PROGRAM r_Gestion_Actionneurs_TOR
VAR
	XV_Alim_Douche: Registre_V1;
	XV_Alim_Douchette: Registre_V1;
	XV_Alim_Lavabo: Registre_V1;
	XV_Vid_Douche: Registre_V1;
	XV_Vid_Lavabo: Registre_V1;
	XV_Electrovanne_Douche: Registre_V1;
	XV_Electrovanne_Lavabo: Registre_V1;
	Prise_Cabine: Prise;
	XV_Vanne_Souf_Bas_Deb: Registre_V1;
	XV_Vanne_Ext_Bas_Deb: Registre_V1;
	Reg_Etanche_Souf: Registre_V1;
	XV_Alim_NEP: Registre_V1;
	Y_Verin_WC_GV: Registre_V1;
	Y_Verin_WC_PV: Registre_V1;
	Gestion_EA_WC: Sontay_4RM;
END_VAR

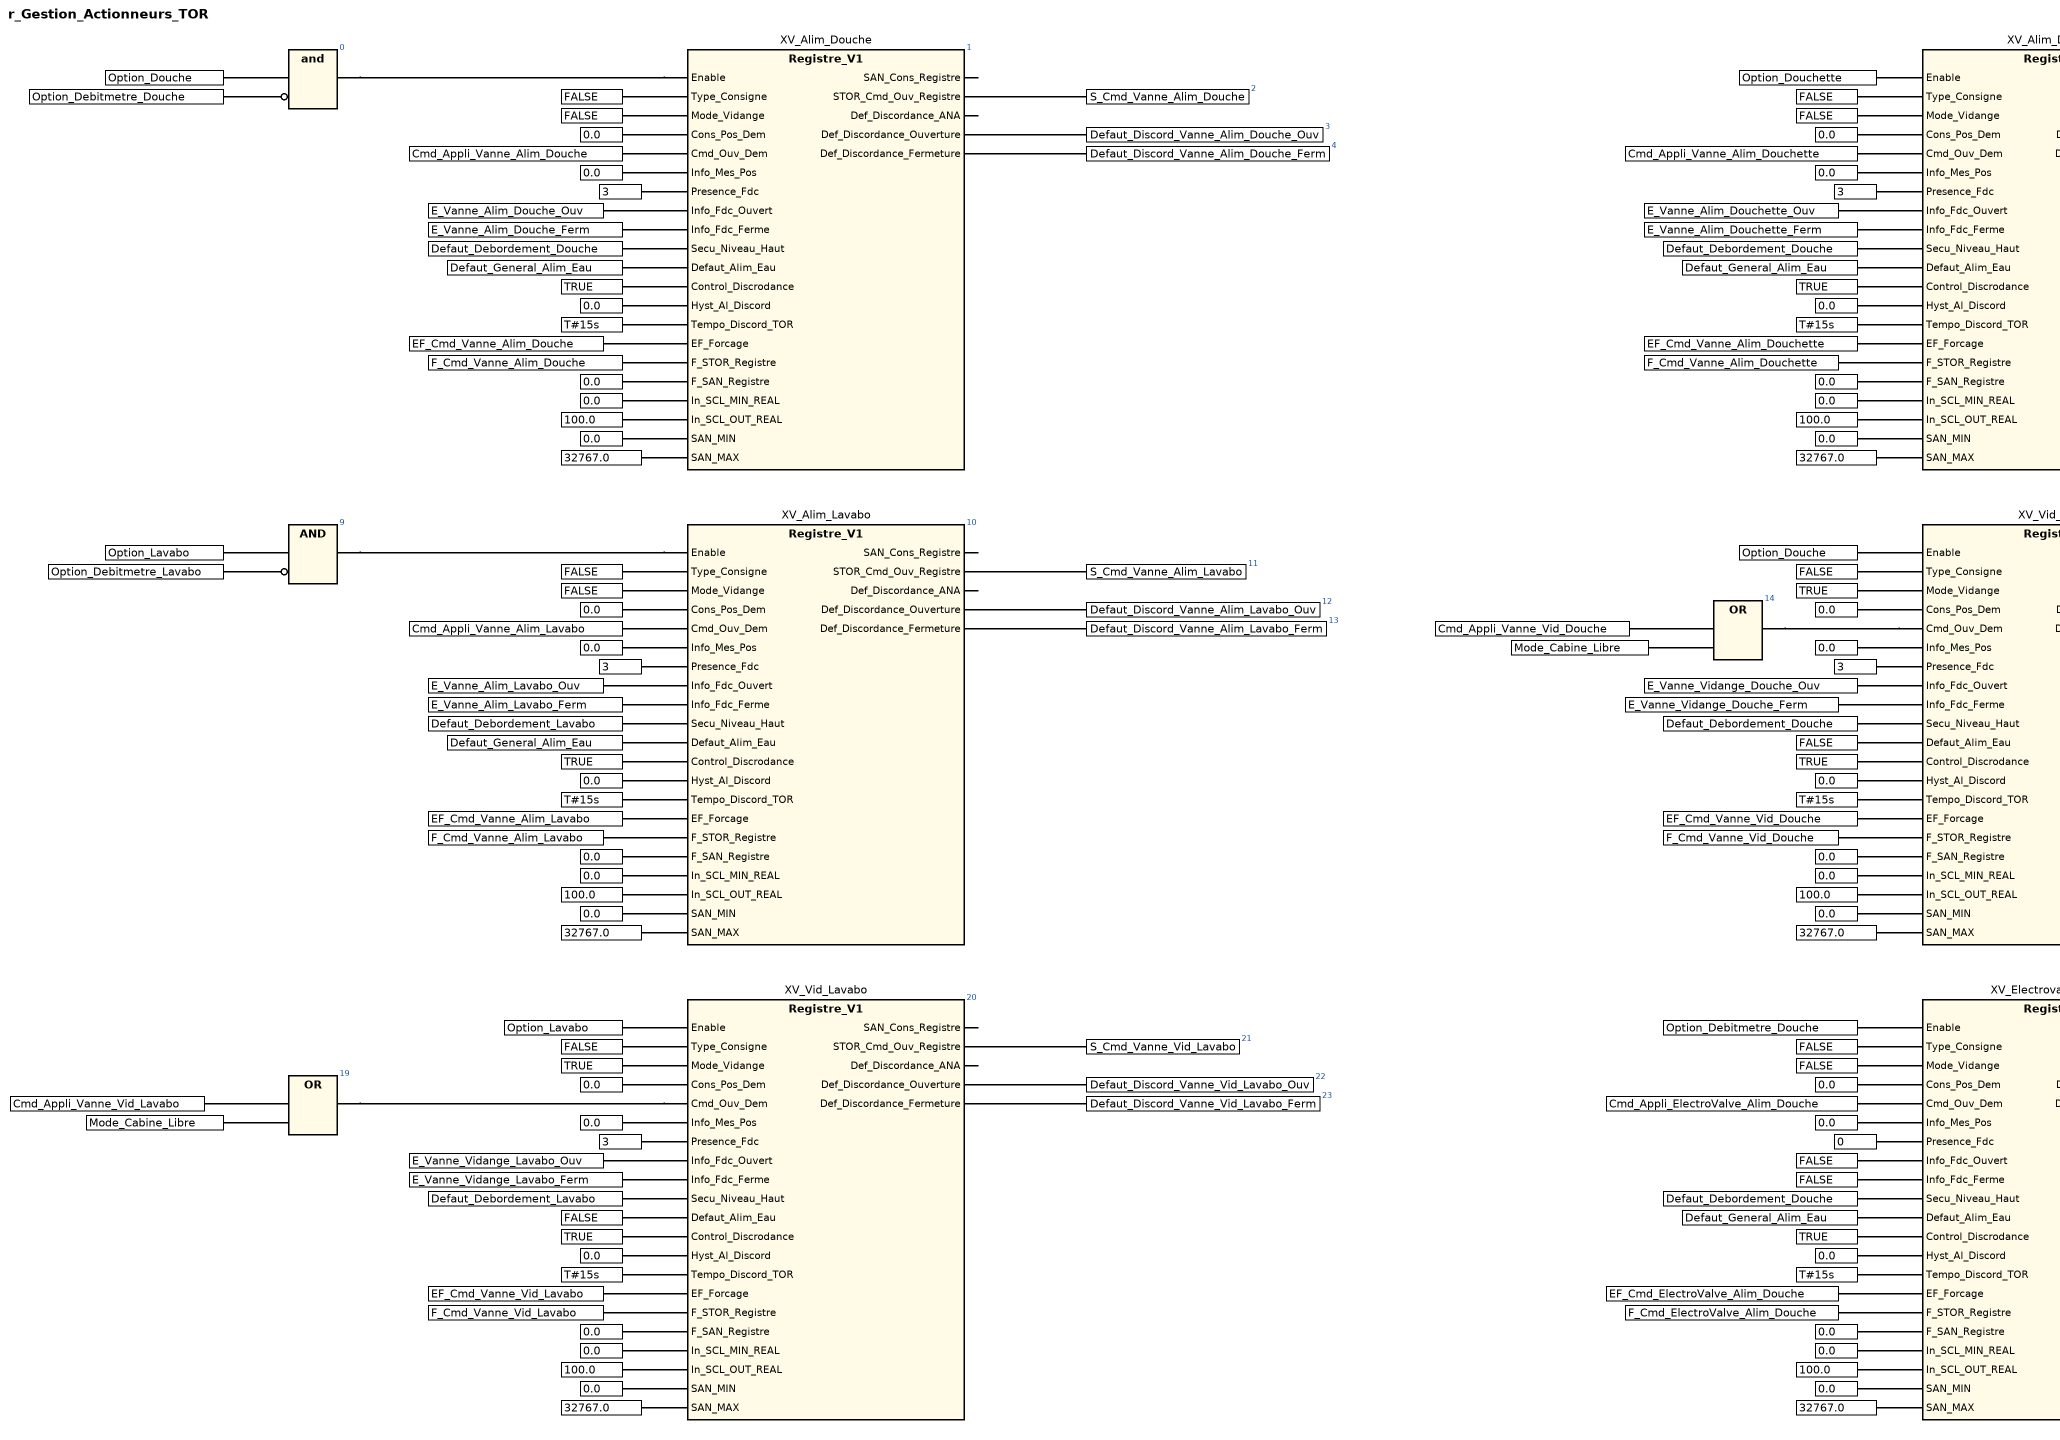
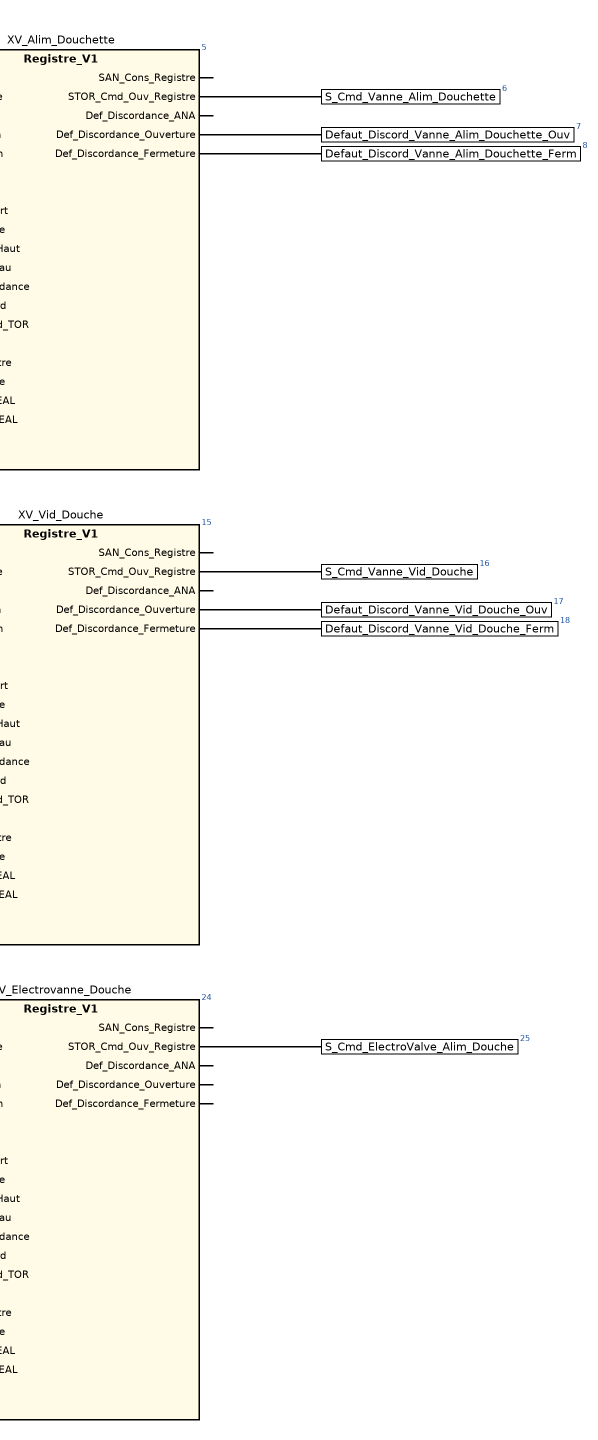
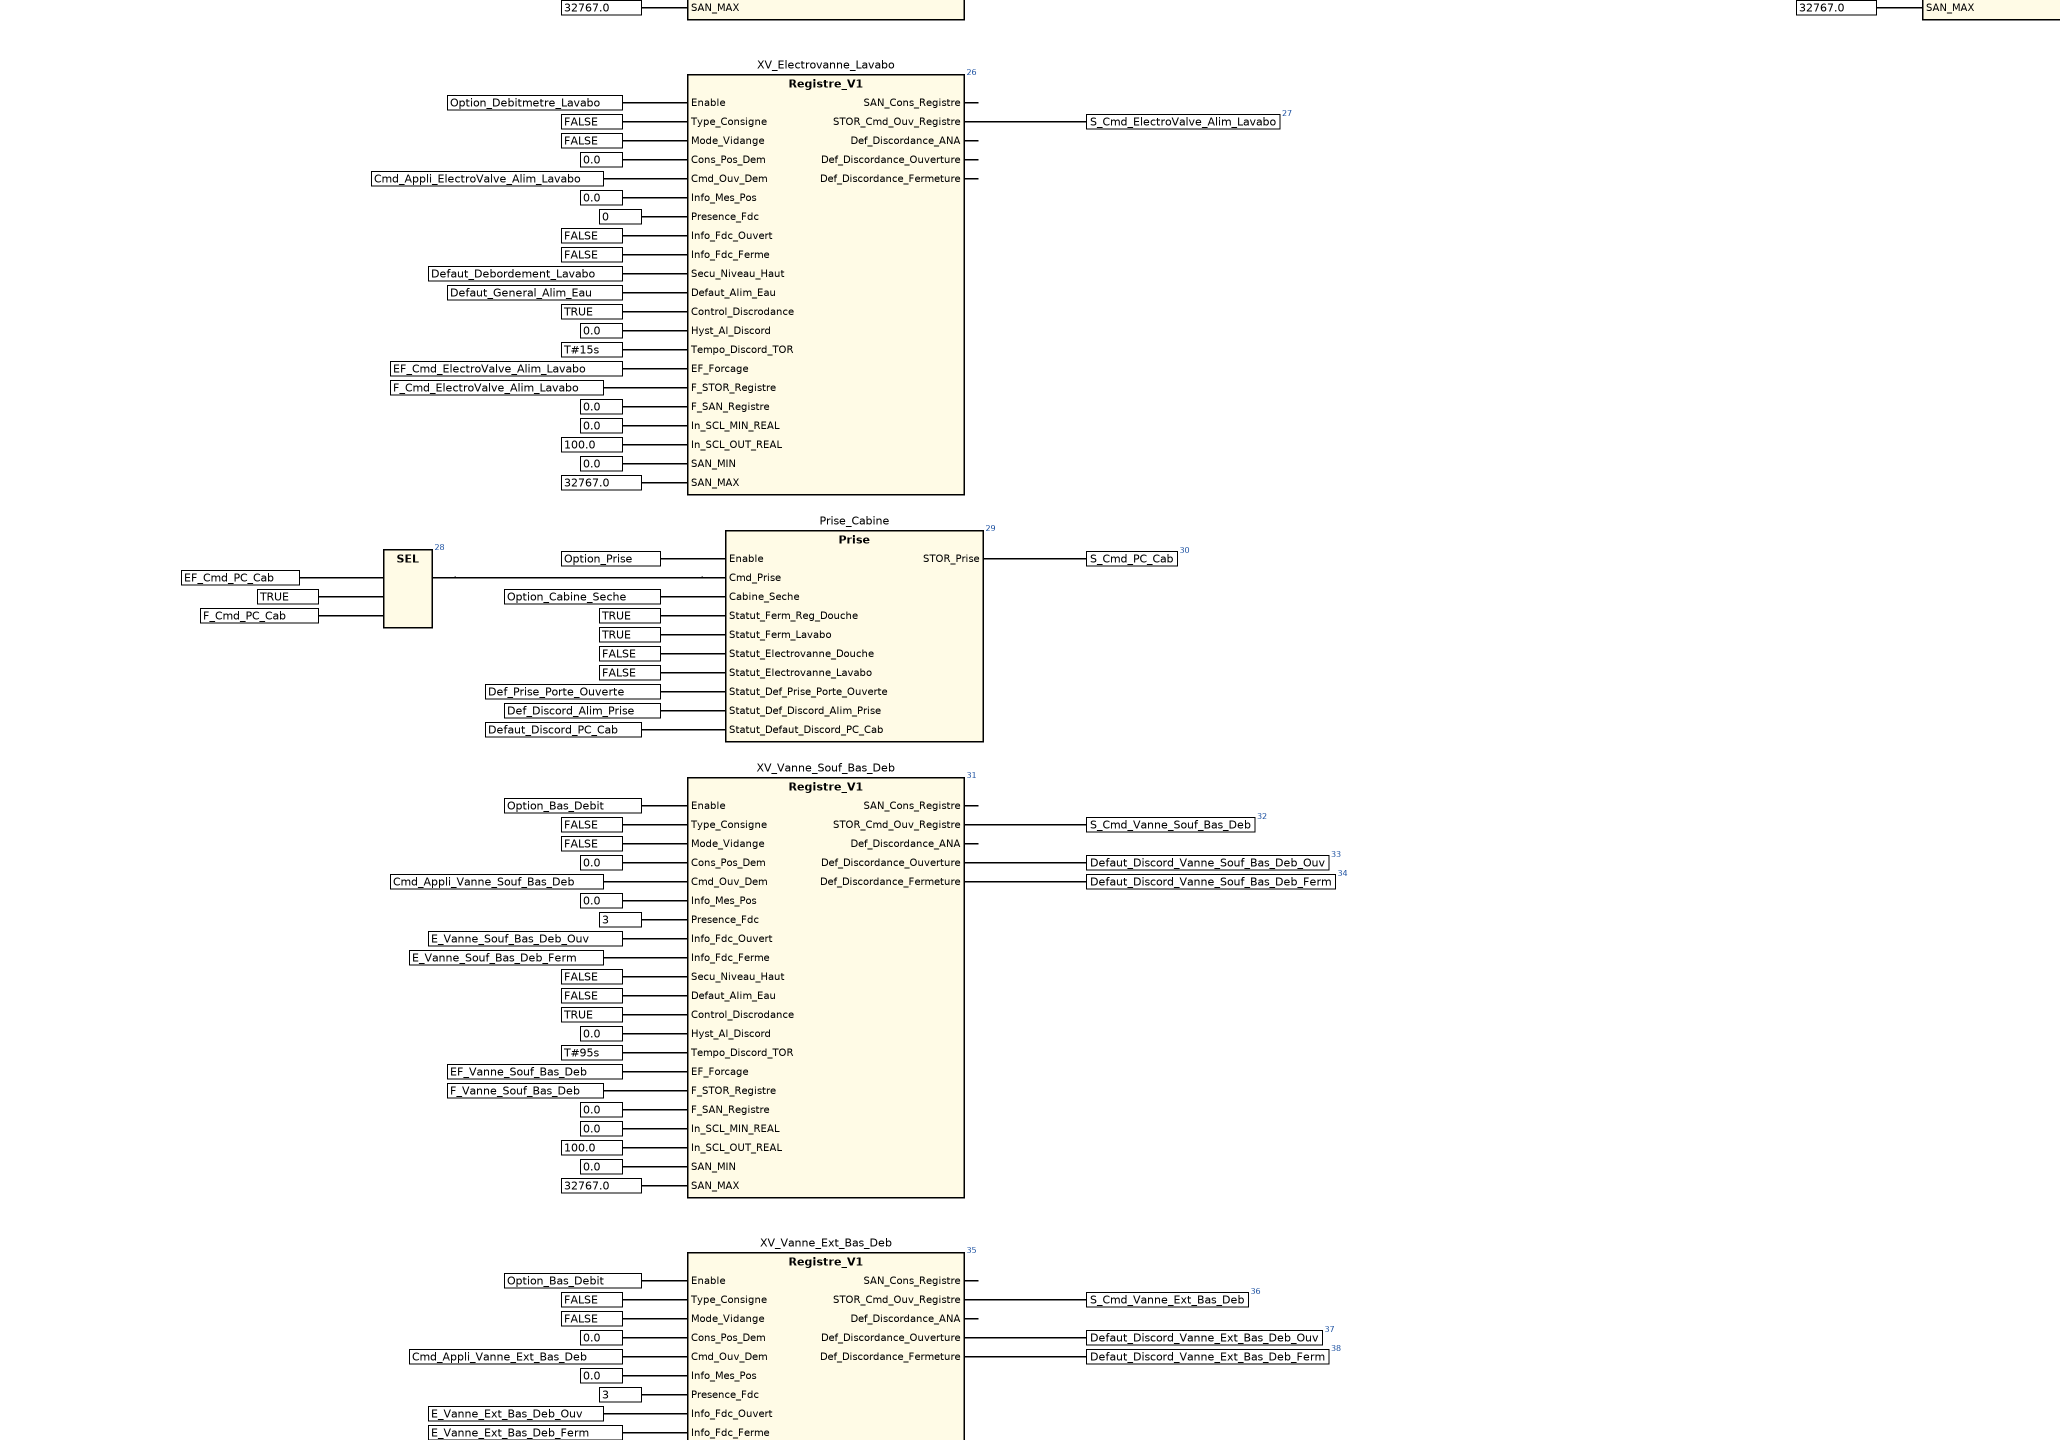
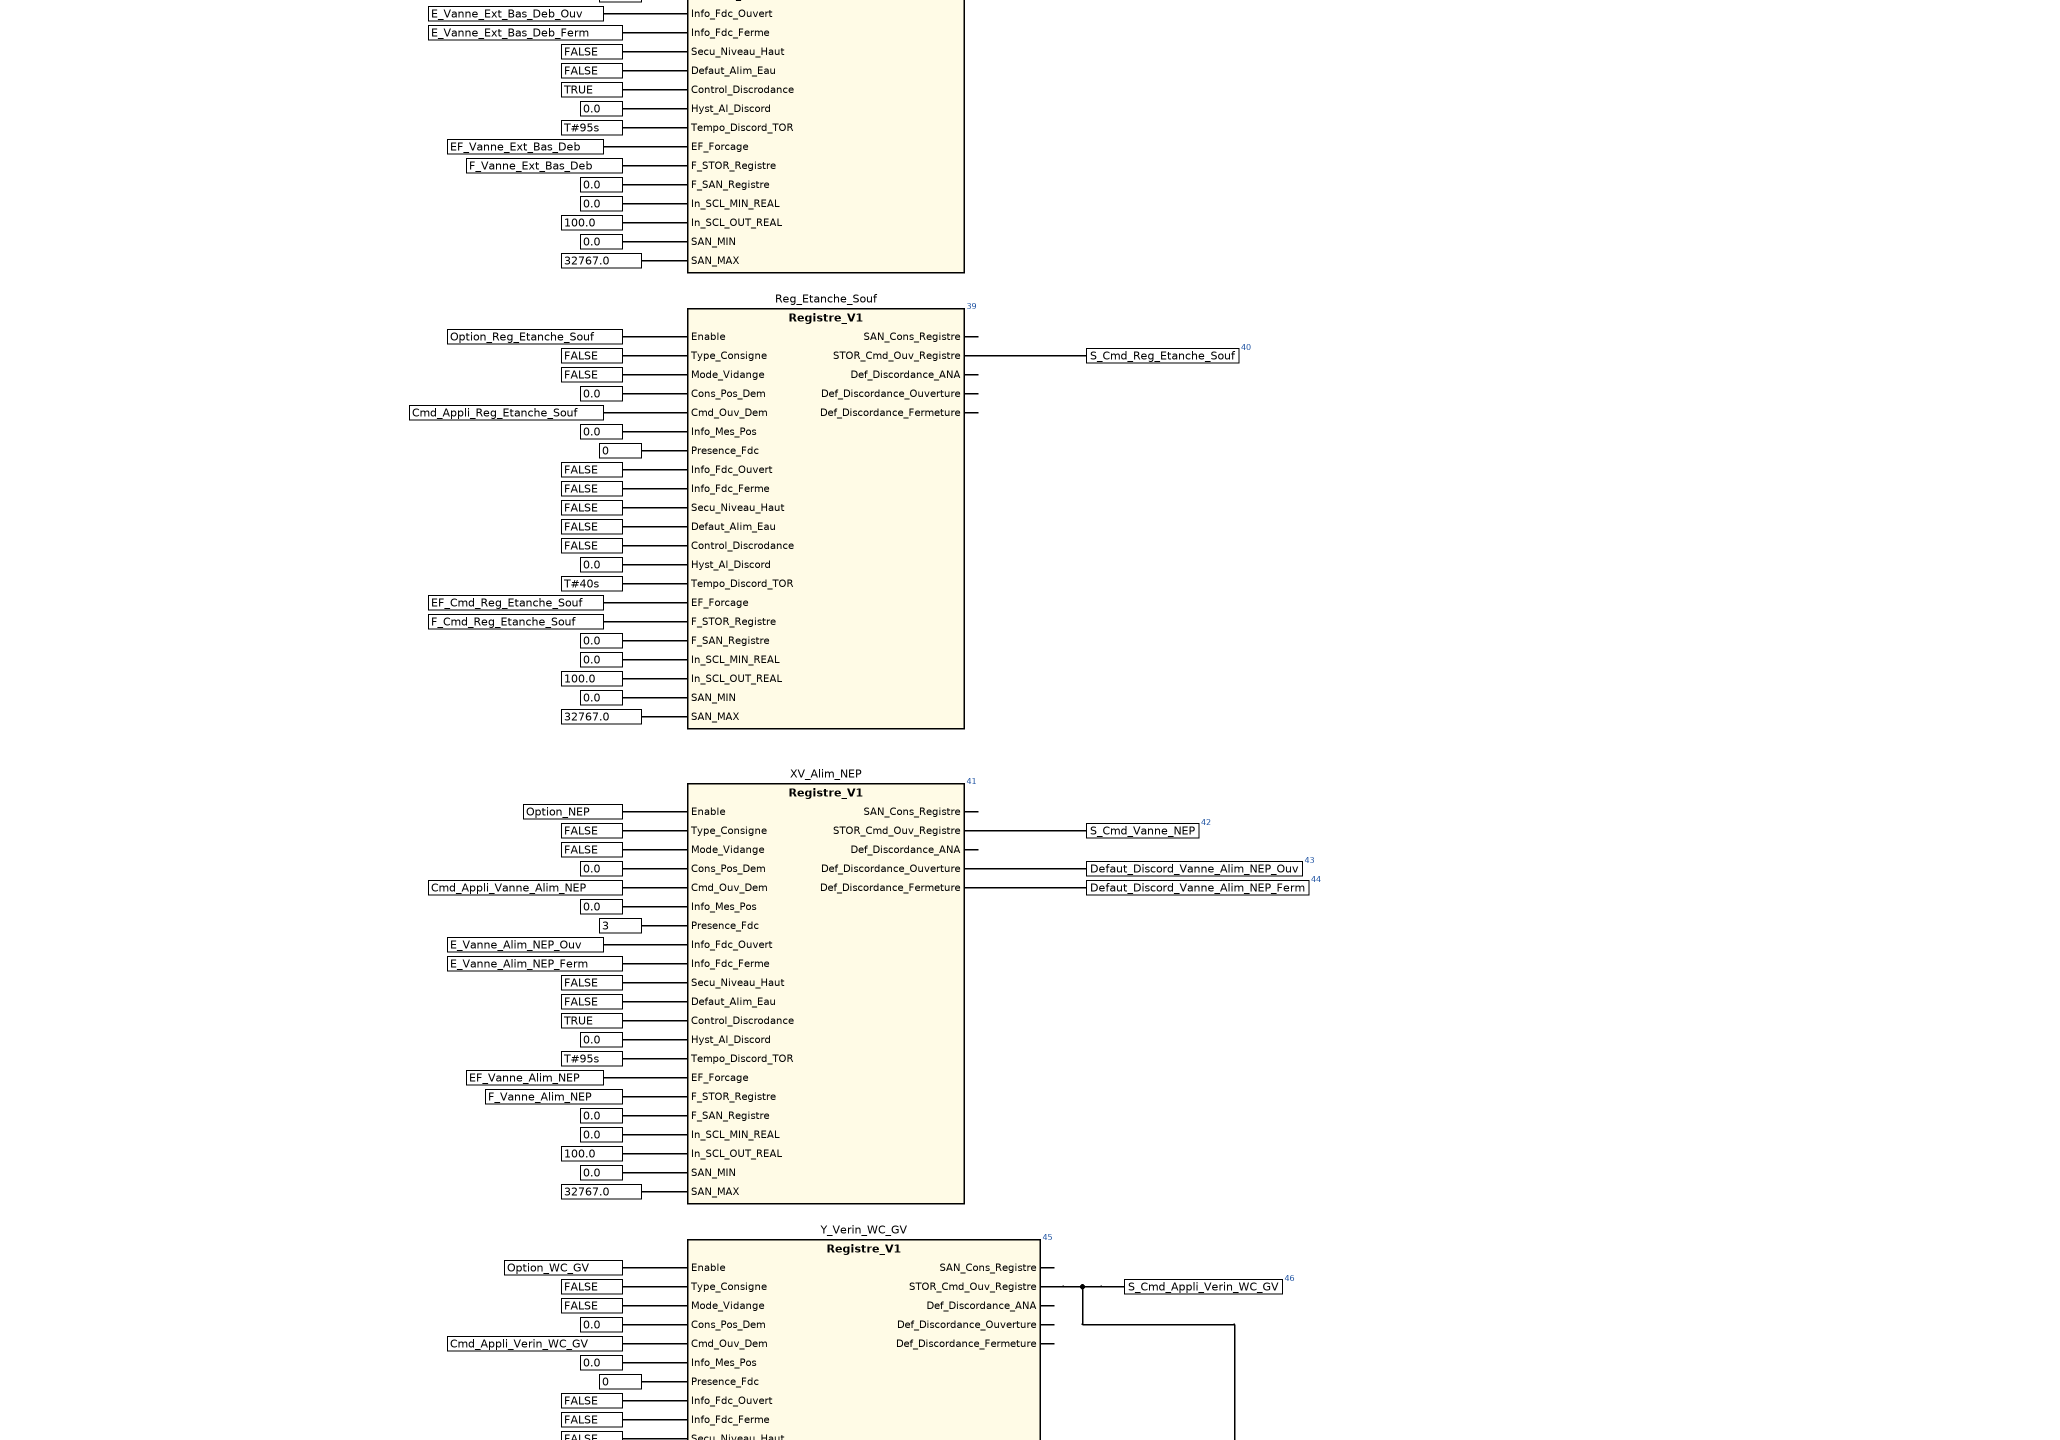
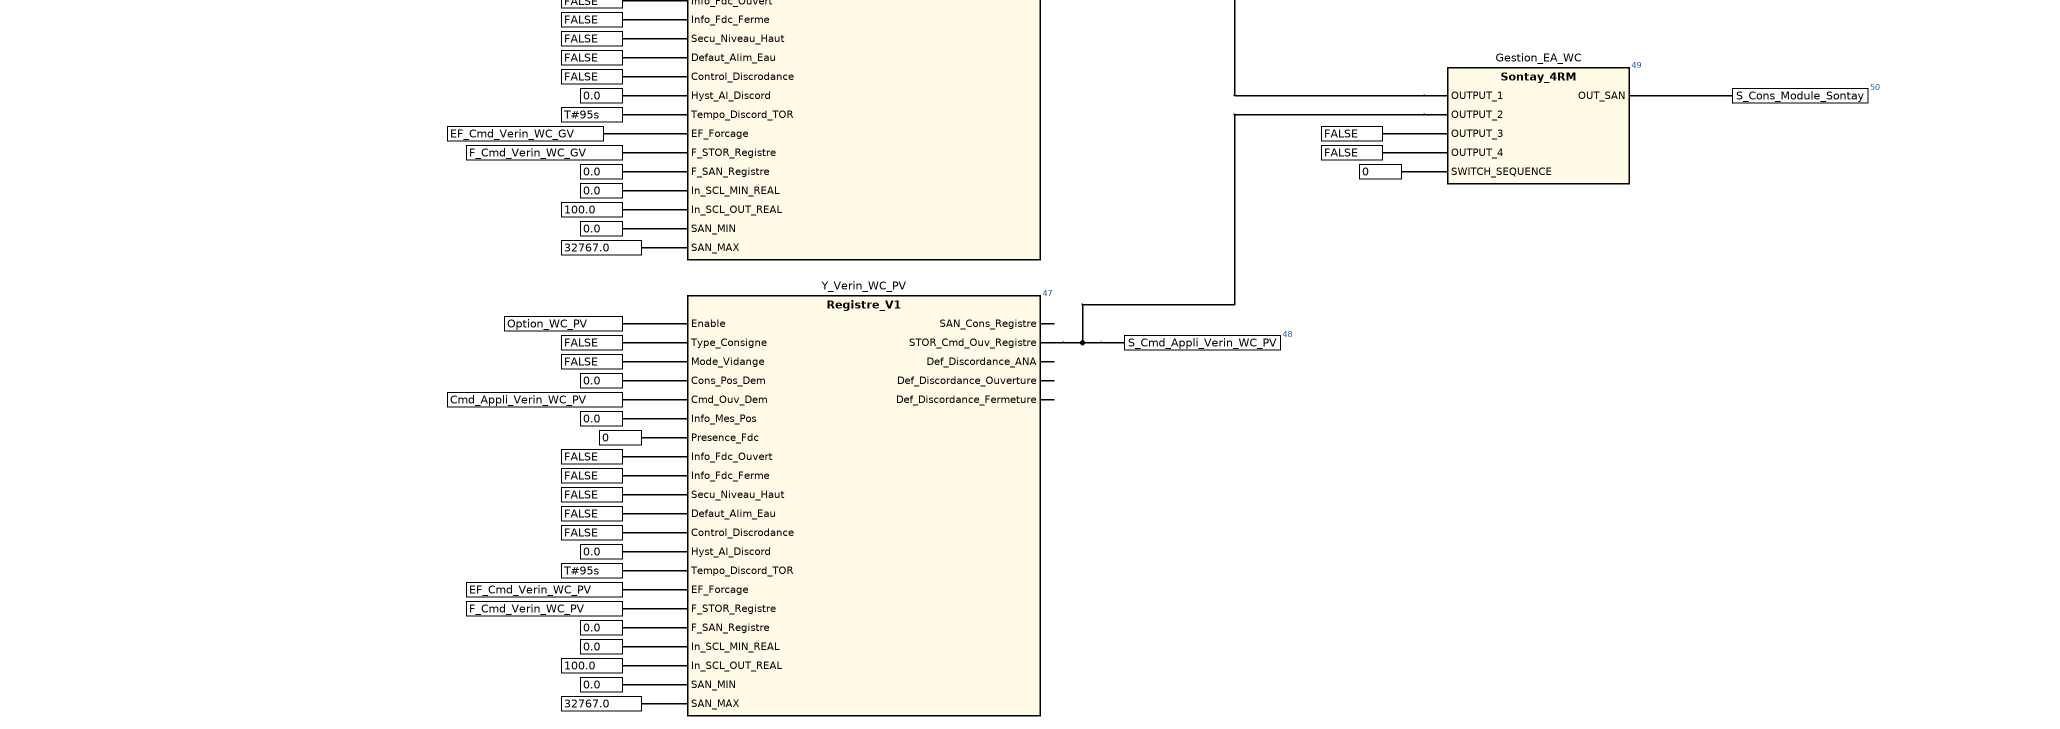
XV_Alim_Douche(
    Enable := Option_Douche AND NOT Option_Debitmetre_Douche,
    Type_Consigne := FALSE,
    Mode_Vidange := FALSE,
    Cons_Pos_Dem := 0.0,
    Cmd_Ouv_Dem := Cmd_Appli_Vanne_Alim_Douche,
    Info_Mes_Pos := 0.0,
    Presence_Fdc := 3,
    Info_Fdc_Ouvert := E_Vanne_Alim_Douche_Ouv,
    Info_Fdc_Ferme := E_Vanne_Alim_Douche_Ferm,
    Secu_Niveau_Haut := Defaut_Debordement_Douche,
    Defaut_Alim_Eau := Defaut_General_Alim_Eau,
    Control_Discrodance := TRUE,
    Hyst_Al_Discord := 0.0,
    Tempo_Discord_TOR := T#15s,
    EF_Forcage := EF_Cmd_Vanne_Alim_Douche,
    F_STOR_Registre := F_Cmd_Vanne_Alim_Douche,
    F_SAN_Registre := 0.0,
    In_SCL_MIN_REAL := 0.0,
    In_SCL_OUT_REAL := 100.0,
    SAN_MIN := 0.0,
    SAN_MAX := 32767.0); // Registre_V1
S_Cmd_Vanne_Alim_Douche := XV_Alim_Douche.STOR_Cmd_Ouv_Registre;
Defaut_Discord_Vanne_Alim_Douche_Ouv := XV_Alim_Douche.Def_Discordance_Ouverture;
Defaut_Discord_Vanne_Alim_Douche_Ferm := XV_Alim_Douche.Def_Discordance_Fermeture;
XV_Alim_Douchette(
    Enable := Option_Douchette,
    Type_Consigne := FALSE,
    Mode_Vidange := FALSE,
    Cons_Pos_Dem := 0.0,
    Cmd_Ouv_Dem := Cmd_Appli_Vanne_Alim_Douchette,
    Info_Mes_Pos := 0.0,
    Presence_Fdc := 3,
    Info_Fdc_Ouvert := E_Vanne_Alim_Douchette_Ouv,
    Info_Fdc_Ferme := E_Vanne_Alim_Douchette_Ferm,
    Secu_Niveau_Haut := Defaut_Debordement_Douche,
    Defaut_Alim_Eau := Defaut_General_Alim_Eau,
    Control_Discrodance := TRUE,
    Hyst_Al_Discord := 0.0,
    Tempo_Discord_TOR := T#15s,
    EF_Forcage := EF_Cmd_Vanne_Alim_Douchette,
    F_STOR_Registre := F_Cmd_Vanne_Alim_Douchette,
    F_SAN_Registre := 0.0,
    In_SCL_MIN_REAL := 0.0,
    In_SCL_OUT_REAL := 100.0,
    SAN_MIN := 0.0,
    SAN_MAX := 32767.0); // Registre_V1
S_Cmd_Vanne_Alim_Douchette := XV_Alim_Douchette.STOR_Cmd_Ouv_Registre;
Defaut_Discord_Vanne_Alim_Douchette_Ouv := XV_Alim_Douchette.Def_Discordance_Ouverture;
Defaut_Discord_Vanne_Alim_Douchette_Ferm := XV_Alim_Douchette.Def_Discordance_Fermeture;
XV_Alim_Lavabo(
    Enable := Option_Lavabo AND NOT Option_Debitmetre_Lavabo,
    Type_Consigne := FALSE,
    Mode_Vidange := FALSE,
    Cons_Pos_Dem := 0.0,
    Cmd_Ouv_Dem := Cmd_Appli_Vanne_Alim_Lavabo,
    Info_Mes_Pos := 0.0,
    Presence_Fdc := 3,
    Info_Fdc_Ouvert := E_Vanne_Alim_Lavabo_Ouv,
    Info_Fdc_Ferme := E_Vanne_Alim_Lavabo_Ferm,
    Secu_Niveau_Haut := Defaut_Debordement_Lavabo,
    Defaut_Alim_Eau := Defaut_General_Alim_Eau,
    Control_Discrodance := TRUE,
    Hyst_Al_Discord := 0.0,
    Tempo_Discord_TOR := T#15s,
    EF_Forcage := EF_Cmd_Vanne_Alim_Lavabo,
    F_STOR_Registre := F_Cmd_Vanne_Alim_Lavabo,
    F_SAN_Registre := 0.0,
    In_SCL_MIN_REAL := 0.0,
    In_SCL_OUT_REAL := 100.0,
    SAN_MIN := 0.0,
    SAN_MAX := 32767.0); // Registre_V1
S_Cmd_Vanne_Alim_Lavabo := XV_Alim_Lavabo.STOR_Cmd_Ouv_Registre;
Defaut_Discord_Vanne_Alim_Lavabo_Ouv := XV_Alim_Lavabo.Def_Discordance_Ouverture;
Defaut_Discord_Vanne_Alim_Lavabo_Ferm := XV_Alim_Lavabo.Def_Discordance_Fermeture;
XV_Vid_Douche(
    Enable := Option_Douche,
    Type_Consigne := FALSE,
    Mode_Vidange := TRUE,
    Cons_Pos_Dem := 0.0,
    Cmd_Ouv_Dem := Cmd_Appli_Vanne_Vid_Douche OR Mode_Cabine_Libre,
    Info_Mes_Pos := 0.0,
    Presence_Fdc := 3,
    Info_Fdc_Ouvert := E_Vanne_Vidange_Douche_Ouv,
    Info_Fdc_Ferme := E_Vanne_Vidange_Douche_Ferm,
    Secu_Niveau_Haut := Defaut_Debordement_Douche,
    Defaut_Alim_Eau := FALSE,
    Control_Discrodance := TRUE,
    Hyst_Al_Discord := 0.0,
    Tempo_Discord_TOR := T#15s,
    EF_Forcage := EF_Cmd_Vanne_Vid_Douche,
    F_STOR_Registre := F_Cmd_Vanne_Vid_Douche,
    F_SAN_Registre := 0.0,
    In_SCL_MIN_REAL := 0.0,
    In_SCL_OUT_REAL := 100.0,
    SAN_MIN := 0.0,
    SAN_MAX := 32767.0); // Registre_V1
S_Cmd_Vanne_Vid_Douche := XV_Vid_Douche.STOR_Cmd_Ouv_Registre;
Defaut_Discord_Vanne_Vid_Douche_Ouv := XV_Vid_Douche.Def_Discordance_Ouverture;
Defaut_Discord_Vanne_Vid_Douche_Ferm := XV_Vid_Douche.Def_Discordance_Fermeture;
XV_Vid_Lavabo(
    Enable := Option_Lavabo,
    Type_Consigne := FALSE,
    Mode_Vidange := TRUE,
    Cons_Pos_Dem := 0.0,
    Cmd_Ouv_Dem := Cmd_Appli_Vanne_Vid_Lavabo OR Mode_Cabine_Libre,
    Info_Mes_Pos := 0.0,
    Presence_Fdc := 3,
    Info_Fdc_Ouvert := E_Vanne_Vidange_Lavabo_Ouv,
    Info_Fdc_Ferme := E_Vanne_Vidange_Lavabo_Ferm,
    Secu_Niveau_Haut := Defaut_Debordement_Lavabo,
    Defaut_Alim_Eau := FALSE,
    Control_Discrodance := TRUE,
    Hyst_Al_Discord := 0.0,
    Tempo_Discord_TOR := T#15s,
    EF_Forcage := EF_Cmd_Vanne_Vid_Lavabo,
    F_STOR_Registre := F_Cmd_Vanne_Vid_Lavabo,
    F_SAN_Registre := 0.0,
    In_SCL_MIN_REAL := 0.0,
    In_SCL_OUT_REAL := 100.0,
    SAN_MIN := 0.0,
    SAN_MAX := 32767.0); // Registre_V1
S_Cmd_Vanne_Vid_Lavabo := XV_Vid_Lavabo.STOR_Cmd_Ouv_Registre;
Defaut_Discord_Vanne_Vid_Lavabo_Ouv := XV_Vid_Lavabo.Def_Discordance_Ouverture;
Defaut_Discord_Vanne_Vid_Lavabo_Ferm := XV_Vid_Lavabo.Def_Discordance_Fermeture;
XV_Electrovanne_Douche(
    Enable := Option_Debitmetre_Douche,
    Type_Consigne := FALSE,
    Mode_Vidange := FALSE,
    Cons_Pos_Dem := 0.0,
    Cmd_Ouv_Dem := Cmd_Appli_ElectroValve_Alim_Douche,
    Info_Mes_Pos := 0.0,
    Presence_Fdc := 0,
    Info_Fdc_Ouvert := FALSE,
    Info_Fdc_Ferme := FALSE,
    Secu_Niveau_Haut := Defaut_Debordement_Douche,
    Defaut_Alim_Eau := Defaut_General_Alim_Eau,
    Control_Discrodance := TRUE,
    Hyst_Al_Discord := 0.0,
    Tempo_Discord_TOR := T#15s,
    EF_Forcage := EF_Cmd_ElectroValve_Alim_Douche,
    F_STOR_Registre := F_Cmd_ElectroValve_Alim_Douche,
    F_SAN_Registre := 0.0,
    In_SCL_MIN_REAL := 0.0,
    In_SCL_OUT_REAL := 100.0,
    SAN_MIN := 0.0,
    SAN_MAX := 32767.0); // Registre_V1
S_Cmd_ElectroValve_Alim_Douche := XV_Electrovanne_Douche.STOR_Cmd_Ouv_Registre;
XV_Electrovanne_Lavabo(
    Enable := Option_Debitmetre_Lavabo,
    Type_Consigne := FALSE,
    Mode_Vidange := FALSE,
    Cons_Pos_Dem := 0.0,
    Cmd_Ouv_Dem := Cmd_Appli_ElectroValve_Alim_Lavabo,
    Info_Mes_Pos := 0.0,
    Presence_Fdc := 0,
    Info_Fdc_Ouvert := FALSE,
    Info_Fdc_Ferme := FALSE,
    Secu_Niveau_Haut := Defaut_Debordement_Lavabo,
    Defaut_Alim_Eau := Defaut_General_Alim_Eau,
    Control_Discrodance := TRUE,
    Hyst_Al_Discord := 0.0,
    Tempo_Discord_TOR := T#15s,
    EF_Forcage := EF_Cmd_ElectroValve_Alim_Lavabo,
    F_STOR_Registre := F_Cmd_ElectroValve_Alim_Lavabo,
    F_SAN_Registre := 0.0,
    In_SCL_MIN_REAL := 0.0,
    In_SCL_OUT_REAL := 100.0,
    SAN_MIN := 0.0,
    SAN_MAX := 32767.0); // Registre_V1
S_Cmd_ElectroValve_Alim_Lavabo := XV_Electrovanne_Lavabo.STOR_Cmd_Ouv_Registre;
Prise_Cabine(
    Enable := Option_Prise,
    Cmd_Prise := SEL(EF_Cmd_PC_Cab, TRUE, F_Cmd_PC_Cab),
    Cabine_Seche := Option_Cabine_Seche,
    Statut_Ferm_Reg_Douche := TRUE,
    Statut_Ferm_Lavabo := TRUE,
    Statut_Electrovanne_Douche := FALSE,
    Statut_Electrovanne_Lavabo := FALSE,
    Statut_Def_Prise_Porte_Ouverte := Def_Prise_Porte_Ouverte,
    Statut_Def_Discord_Alim_Prise := Def_Discord_Alim_Prise,
    Statut_Defaut_Discord_PC_Cab := Defaut_Discord_PC_Cab); // Prise
S_Cmd_PC_Cab := Prise_Cabine.STOR_Prise;
XV_Vanne_Souf_Bas_Deb(
    Enable := Option_Bas_Debit,
    Type_Consigne := FALSE,
    Mode_Vidange := FALSE,
    Cons_Pos_Dem := 0.0,
    Cmd_Ouv_Dem := Cmd_Appli_Vanne_Souf_Bas_Deb,
    Info_Mes_Pos := 0.0,
    Presence_Fdc := 3,
    Info_Fdc_Ouvert := E_Vanne_Souf_Bas_Deb_Ouv,
    Info_Fdc_Ferme := E_Vanne_Souf_Bas_Deb_Ferm,
    Secu_Niveau_Haut := FALSE,
    Defaut_Alim_Eau := FALSE,
    Control_Discrodance := TRUE,
    Hyst_Al_Discord := 0.0,
    Tempo_Discord_TOR := T#95s,
    EF_Forcage := EF_Vanne_Souf_Bas_Deb,
    F_STOR_Registre := F_Vanne_Souf_Bas_Deb,
    F_SAN_Registre := 0.0,
    In_SCL_MIN_REAL := 0.0,
    In_SCL_OUT_REAL := 100.0,
    SAN_MIN := 0.0,
    SAN_MAX := 32767.0); // Registre_V1
S_Cmd_Vanne_Souf_Bas_Deb := XV_Vanne_Souf_Bas_Deb.STOR_Cmd_Ouv_Registre;
Defaut_Discord_Vanne_Souf_Bas_Deb_Ouv := XV_Vanne_Souf_Bas_Deb.Def_Discordance_Ouverture;
Defaut_Discord_Vanne_Souf_Bas_Deb_Ferm := XV_Vanne_Souf_Bas_Deb.Def_Discordance_Fermeture;
XV_Vanne_Ext_Bas_Deb(
    Enable := Option_Bas_Debit,
    Type_Consigne := FALSE,
    Mode_Vidange := FALSE,
    Cons_Pos_Dem := 0.0,
    Cmd_Ouv_Dem := Cmd_Appli_Vanne_Ext_Bas_Deb,
    Info_Mes_Pos := 0.0,
    Presence_Fdc := 3,
    Info_Fdc_Ouvert := E_Vanne_Ext_Bas_Deb_Ouv,
    Info_Fdc_Ferme := E_Vanne_Ext_Bas_Deb_Ferm,
    Secu_Niveau_Haut := FALSE,
    Defaut_Alim_Eau := FALSE,
    Control_Discrodance := TRUE,
    Hyst_Al_Discord := 0.0,
    Tempo_Discord_TOR := T#95s,
    EF_Forcage := EF_Vanne_Ext_Bas_Deb,
    F_STOR_Registre := F_Vanne_Ext_Bas_Deb,
    F_SAN_Registre := 0.0,
    In_SCL_MIN_REAL := 0.0,
    In_SCL_OUT_REAL := 100.0,
    SAN_MIN := 0.0,
    SAN_MAX := 32767.0); // Registre_V1
S_Cmd_Vanne_Ext_Bas_Deb := XV_Vanne_Ext_Bas_Deb.STOR_Cmd_Ouv_Registre;
Defaut_Discord_Vanne_Ext_Bas_Deb_Ouv := XV_Vanne_Ext_Bas_Deb.Def_Discordance_Ouverture;
Defaut_Discord_Vanne_Ext_Bas_Deb_Ferm := XV_Vanne_Ext_Bas_Deb.Def_Discordance_Fermeture;
Reg_Etanche_Souf(
    Enable := Option_Reg_Etanche_Souf,
    Type_Consigne := FALSE,
    Mode_Vidange := FALSE,
    Cons_Pos_Dem := 0.0,
    Cmd_Ouv_Dem := Cmd_Appli_Reg_Etanche_Souf,
    Info_Mes_Pos := 0.0,
    Presence_Fdc := 0,
    Info_Fdc_Ouvert := FALSE,
    Info_Fdc_Ferme := FALSE,
    Secu_Niveau_Haut := FALSE,
    Defaut_Alim_Eau := FALSE,
    Control_Discrodance := FALSE,
    Hyst_Al_Discord := 0.0,
    Tempo_Discord_TOR := T#40s,
    EF_Forcage := EF_Cmd_Reg_Etanche_Souf,
    F_STOR_Registre := F_Cmd_Reg_Etanche_Souf,
    F_SAN_Registre := 0.0,
    In_SCL_MIN_REAL := 0.0,
    In_SCL_OUT_REAL := 100.0,
    SAN_MIN := 0.0,
    SAN_MAX := 32767.0); // Registre_V1
S_Cmd_Reg_Etanche_Souf := Reg_Etanche_Souf.STOR_Cmd_Ouv_Registre;
XV_Alim_NEP(
    Enable := Option_NEP,
    Type_Consigne := FALSE,
    Mode_Vidange := FALSE,
    Cons_Pos_Dem := 0.0,
    Cmd_Ouv_Dem := Cmd_Appli_Vanne_Alim_NEP,
    Info_Mes_Pos := 0.0,
    Presence_Fdc := 3,
    Info_Fdc_Ouvert := E_Vanne_Alim_NEP_Ouv,
    Info_Fdc_Ferme := E_Vanne_Alim_NEP_Ferm,
    Secu_Niveau_Haut := FALSE,
    Defaut_Alim_Eau := FALSE,
    Control_Discrodance := TRUE,
    Hyst_Al_Discord := 0.0,
    Tempo_Discord_TOR := T#95s,
    EF_Forcage := EF_Vanne_Alim_NEP,
    F_STOR_Registre := F_Vanne_Alim_NEP,
    F_SAN_Registre := 0.0,
    In_SCL_MIN_REAL := 0.0,
    In_SCL_OUT_REAL := 100.0,
    SAN_MIN := 0.0,
    SAN_MAX := 32767.0); // Registre_V1
S_Cmd_Vanne_NEP := XV_Alim_NEP.STOR_Cmd_Ouv_Registre;
Defaut_Discord_Vanne_Alim_NEP_Ouv := XV_Alim_NEP.Def_Discordance_Ouverture;
Defaut_Discord_Vanne_Alim_NEP_Ferm := XV_Alim_NEP.Def_Discordance_Fermeture;
Y_Verin_WC_GV(
    Enable := Option_WC_GV,
    Type_Consigne := FALSE,
    Mode_Vidange := FALSE,
    Cons_Pos_Dem := 0.0,
    Cmd_Ouv_Dem := Cmd_Appli_Verin_WC_GV,
    Info_Mes_Pos := 0.0,
    Presence_Fdc := 0,
    Info_Fdc_Ouvert := FALSE,
    Info_Fdc_Ferme := FALSE,
    Secu_Niveau_Haut := FALSE,
    Defaut_Alim_Eau := FALSE,
    Control_Discrodance := FALSE,
    Hyst_Al_Discord := 0.0,
    Tempo_Discord_TOR := T#95s,
    EF_Forcage := EF_Cmd_Verin_WC_GV,
    F_STOR_Registre := F_Cmd_Verin_WC_GV,
    F_SAN_Registre := 0.0,
    In_SCL_MIN_REAL := 0.0,
    In_SCL_OUT_REAL := 100.0,
    SAN_MIN := 0.0,
    SAN_MAX := 32767.0); // Registre_V1
S_Cmd_Appli_Verin_WC_GV := Y_Verin_WC_GV.STOR_Cmd_Ouv_Registre;
Y_Verin_WC_PV(
    Enable := Option_WC_PV,
    Type_Consigne := FALSE,
    Mode_Vidange := FALSE,
    Cons_Pos_Dem := 0.0,
    Cmd_Ouv_Dem := Cmd_Appli_Verin_WC_PV,
    Info_Mes_Pos := 0.0,
    Presence_Fdc := 0,
    Info_Fdc_Ouvert := FALSE,
    Info_Fdc_Ferme := FALSE,
    Secu_Niveau_Haut := FALSE,
    Defaut_Alim_Eau := FALSE,
    Control_Discrodance := FALSE,
    Hyst_Al_Discord := 0.0,
    Tempo_Discord_TOR := T#95s,
    EF_Forcage := EF_Cmd_Verin_WC_PV,
    F_STOR_Registre := F_Cmd_Verin_WC_PV,
    F_SAN_Registre := 0.0,
    In_SCL_MIN_REAL := 0.0,
    In_SCL_OUT_REAL := 100.0,
    SAN_MIN := 0.0,
    SAN_MAX := 32767.0); // Registre_V1
S_Cmd_Appli_Verin_WC_PV := Y_Verin_WC_PV.STOR_Cmd_Ouv_Registre;
Gestion_EA_WC(
    OUTPUT_1 := Y_Verin_WC_GV.STOR_Cmd_Ouv_Registre,
    OUTPUT_2 := Y_Verin_WC_PV.STOR_Cmd_Ouv_Registre,
    OUTPUT_3 := FALSE,
    OUTPUT_4 := FALSE,
    SWITCH_SEQUENCE := 0); // Sontay_4RM
S_Cons_Module_Sontay := Gestion_EA_WC.OUT_SAN;

END_PROGRAM

(* stored: Version 1.1.0.1, ProductVersion 3.1.4024.16
   POU r_Gestion_Actionneurs_TOR: Id {eecb510c-ae44-45ec-a5e3-94a36182441c}, SpecialFunc None *)
